Universal Robots PolyScope program: ability.urp

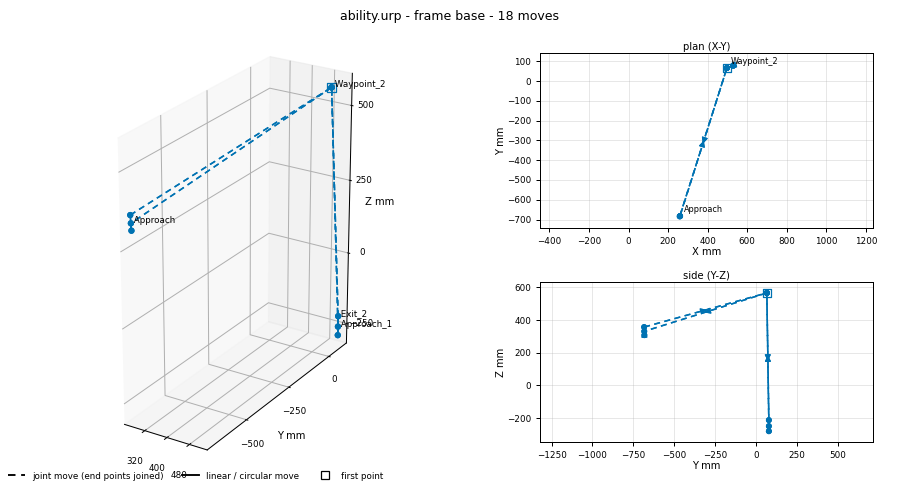
[picture p0: tool path of ability.urp in frame base, 18 of 18 moves have a stored position in this frame; points joined in program order, loops and branches not executed]
Program ability (installation=default directory=/programs createdIn=5.16.0 lastSavedIn=5.21.3 robotSerialNumber=20245590091)
Calibrated DH parameters: a=[0.000082, -0.206079, -0.372164, 0.000031, 0.000055, 0]; d=[0.162506, 220.320261, -282.089171, 61.902297, 0.099578, 0.098999]; alpha=[1.569879, -0.001688, 0.002003, 1.569052, -1.569943, 0]; deltaTheta=[0, -1.064762, 0.743886, 0.320883, 0.000002, 0]
InitVariablesNode variables(variable(name=Pallet_2_cnt_3, expression=1), variable(name=Pallet_2_cnt_4, expression=1), variable(name=Pallet_2_cnt_5, expression=1), variable(name=Pallet_2_cnt_6, expression=1), variable(name=Pallet_2_lct_3, expression=1), variable(name=Pallet_2_lct_4, expression=1), variable(name=Pallet_2_lct_5, expression=1), variable(name=Pallet_2_lct_6, expression=1), variable(name=Pallet_2_lno_3, expression=1), variable(name=Pallet_2_lno_4, expression=1), variable(name=Pallet_2_lno_5, expression=1), variable(name=Pallet_2_lno_6, expression=1), variable(name=Pallet_2_sep_3, expression=False), variable(name=Pallet_2_sep_4, expression=False), variable(name=Pallet_2_sep_5, expression=False), variable(name=Pallet_2_sep_6, expression=False), variable(name=Pallet_2_tct_3, expression=1), variable(name=Pallet_2_tct_4, expression=1), variable(name=Pallet_2_tct_5, expression=1), variable(name=Pallet_2_tct_6, expression=1), variable(name=qNearApproach, expression=[0,0,0,0,0,0]), variable(name=qNearApproach_1, expression=[0,0,0,0,0,0]), variable(name=qNearApproach_2, expression=[0,0,0,0,0,0]), variable(name=qNearApproach_3, expression=[0,0,0,0,0,0]))
Robot Program (runOnlyOnce=false)
  SafeHome (positionOptionType=SPEED_AND_ACCELERATION speed=1.047198 acceleration=1.396263 nextMotionTime=2)
  URCap ER-Ability (EnabledRobotics - ER-ABILITY, Enabled Robotics ApS)
    URCap EventNode (EnabledRobotics - ER-ABILITY, Enabled Robotics ApS) dataModel(er_eventnode_inpname=GripOpen, er_eventnode_retvalname=none)
      URCap Gripper (Robotiq_Grippers, Robotiq Inc.) dataModel(position=0.0, force=100.0, speed=100.0, positionInDouble=0.0, forceInDouble=100.0, speedInDouble=100.0, slaveIds=[9], blocking=true)
    URCap EventNode (EnabledRobotics - ER-ABILITY, Enabled Robotics ApS) dataModel(er_eventnode_inpname=GripClosed, er_eventnode_retvalname=none)
      URCap Gripper (Robotiq_Grippers, Robotiq Inc.) dataModel(position=100.0, force=70.0, speed=100.0, positionInDouble=100.0, forceInDouble=70.0, speedInDouble=100.0, slaveIds=[9], blocking=true)
    URCap EventNode (EnabledRobotics - ER-ABILITY, Enabled Robotics ApS) dataModel(er_eventnode_inpname=Unload, er_eventnode_retvalname=none, er_eventnode_input_arg_names=[arg_pose], er_eventnode_input_arg_types=[pose])
      Unload_ref := __er_Unload_arg_pose
      MoveJ speed 60 deg/s, acceleration 80 deg/s^2 (useActiveTCP=true optimoveEnabled=false optiMoveSpeed=0.3 optiMoveAcceleration=0.09) feature=Base
        Waypoint Waypoint_2: TCP in base x=497.545 y=66.443 z=565.568 mm, rx=2.1662 ry=-2.097 rz=-0.0588 rad; joints [173.064, -87.949, 75.071, -70.913, -94.278, -8.478] deg
      URCap Palletizing (polyscope-pallet-impl, Universal Robots) dataModel(palletFeature=Base, isPalletizing=true, Length(key=objectHeight value=0.02 unit=M), Variable(key=qNearApproach, variable(name=qNearApproach_1, initializeExpression=[0,0,0,0,0,0])), Variable(key=name, variable(name=Pallet_5)), Variable(key=globalCountingVariable, variable(name=Pallet_2_cnt_6, initializeExpression=1)), Variable(key=layerCountingVariable, variable(name=Pallet_2_lct_6, initializeExpression=1)), Variable(key=layerNumberVariable, variable(name=Pallet_2_lno_6, initializeExpression=1)), Variable(key=handleSeparatorVariable, variable(name=Pallet_2_sep_6, initializeExpression=False)), Variable(key=totalCountVariable, variable(name=Pallet_2_tct_6, initializeExpression=1)), Variable(key=referencePoint, variable(featureName=referencePoin_1)), Variable(key=separatorPoint, variable(featureName=separatorPoin_1))); state(isChildrenLocked=true)
        URCap Patterns (polyscope-pallet-impl, Universal Robots) state(isChildrenLocked=true)
          URCap Pattern (polyscope-pallet-impl, Universal Robots) dataModel(UUID=a5dc391e-8dfa-4d41-8d42-d1a3ee492412, patternType=LINE, objects=3, Variable(key=nameVariable, variable(name=Line_Pattern_7))); state(isChildrenLocked=true)
            URCap Item (polyscope-pallet-impl, Universal Robots) dataModel(UUID=72ff3311-31d3-41c2-b996-3017bdb4fd84, patternType=LINE, index=0, calibrationDeltaTheta=[-1.5094818129821053E-8, -1.0647624878232371, 0.7438857393498214, 0.32088328103969005, 1.7447632748163189E-6, 3.439939232040279E-7], calibrationA=[8.193426020278456E-5, -0.2060785642550941, -0.3721635571632287, 3.0822330236917175E-5, 5.5236874526065846E-5, 0.0], calibrationD=[0.1625058419451979, 220.32026122990015, -282.0891711692004, 61.90229668578863, 0.09957797525715827, 0.09899883734970352], calibrationAlpha=[1.569878535244303, -0.0016878983510277897, 0.002002552910479703, 1.5690521837938194, -1.5699432474464643, 0.0], calibrationJointChecksum=[-1471040491, -1470094786, -1472279970, -1460232730, -1457493897, -1460320911], calibrationStatus=2, calibrationValidChecksum=true, baseToFeature=[0.0, 0.0, 0.0, 0.0, 0.0, 0.0], TCPOffset=[-1.9242631868060522E-6, -1.9505851089895998E-7, -4.2845847764150236E-6, -5.771534998269337E-6, -3.203463145879142E-5, 1.411217115060646E-5], JointPositions(key=jointpositions, JointPosition(key=[1], Angle(key=pos value=3.039745 unit=RAD)), JointPosition(key=[2], Angle(key=pos value=-0.112207 unit=RAD)), JointPosition(key=[3], Angle(key=pos value=1.692084 unit=RAD)), JointPosition(key=[4], Angle(key=pos value=-3.160784 unit=RAD)), JointPosition(key=[5], Angle(key=pos value=-1.59557 unit=RAD)), JointPosition(key=[6], Angle(key=pos value=-0.133127 unit=RAD))), Variable(key=variable, variable(name=StartItem_7)))
            URCap Item (polyscope-pallet-impl, Universal Robots) dataModel(UUID=58fef9f4-1789-42d8-bc72-cd3fccb1f7d0, patternType=LINE, index=1, calibrationDeltaTheta=[-1.5094818129821053E-8, -1.0647624878232371, 0.7438857393498214, 0.32088328103969005, 1.7447632748163189E-6, 3.439939232040279E-7], calibrationA=[8.193426020278456E-5, -0.2060785642550941, -0.3721635571632287, 3.0822330236917175E-5, 5.5236874526065846E-5, 0.0], calibrationD=[0.1625058419451979, 220.32026122990015, -282.0891711692004, 61.90229668578863, 0.09957797525715827, 0.09899883734970352], calibrationAlpha=[1.569878535244303, -0.0016878983510277897, 0.002002552910479703, 1.5690521837938194, -1.5699432474464643, 0.0], calibrationJointChecksum=[-1471040491, -1470094786, -1472279970, -1460232730, -1457493897, -1460320911], calibrationStatus=2, calibrationValidChecksum=true, baseToFeature=[0.0, 0.0, 0.0, 0.0, 0.0, 0.0], TCPOffset=[6.884421240790917E-6, -1.3788864439701065E-5, -2.2303486297114983E-5, 3.976905791947326E-5, -9.131492742263298E-6, 1.144757581185306E-5], JointPositions(key=jointpositions, JointPosition(key=[1], Angle(key=pos value=2.706754 unit=RAD)), JointPosition(key=[2], Angle(key=pos value=-0.110768 unit=RAD)), JointPosition(key=[3], Angle(key=pos value=1.673712 unit=RAD)), JointPosition(key=[4], Angle(key=pos value=-3.151042 unit=RAD)), JointPosition(key=[5], Angle(key=pos value=-1.590635 unit=RAD)), JointPosition(key=[6], Angle(key=pos value=-0.466181 unit=RAD))), Variable(key=variable, variable(name=EndItem_7)))
        URCap Layers (polyscope-pallet-impl, Universal Robots) dataModel(separators=[false], selectedPatterns=[a5dc391e-8dfa-4d41-8d42-d1a3ee492412])
        URCap At Each Item (polyscope-pallet-impl, Universal Robots) dataModel(selectedPattern=a5dc391e-8dfa-4d41-8d42-d1a3ee492412, selectedPosition=72ff3311-31d3-41c2-b996-3017bdb4fd84, Approach_calibrationDeltaTheta=[-1.5094818129821053E-8, -1.0647624878232371, 0.7438857393498214, 0.32088328103969005, 1.7447632748163189E-6, 3.439939232040279E-7], Approach_calibrationA=[8.193426020278456E-5, -0.2060785642550941, -0.3721635571632287, 3.0822330236917175E-5, 5.5236874526065846E-5, 0.0], Approach_calibrationD=[0.1625058419451979, 220.32026122990015, -282.0891711692004, 61.90229668578863, 0.09957797525715827, 0.09899883734970352], Approach_calibrationAlpha=[1.569878535244303, -0.0016878983510277897, 0.002002552910479703, 1.5690521837938194, -1.5699432474464643, 0.0], Approach_calibrationJointChecksum=[-1471040491, -1470094786, -1472279970, -1460232730, -1457493897, -1460320911], Approach_calibrationStatus=2, Approach_calibrationValidChecksum=true, Approach_baseToFeature=[0.0, 0.0, 0.0, 0.0, 0.0, 0.0], Approach_TCPOffset=[-1.1739771630381313E-6, -5.9013202938773546E-6, 4.731632657406504E-6, 9.46543669298376E-6, -7.291023009343288E-6, -4.926571632538777E-6], Exit_calibrationDeltaTheta=[-1.5094818129821053E-8, -1.0647624878232371, 0.7438857393498214, 0.32088328103969005, 1.7447632748163189E-6, 3.439939232040279E-7], Exit_calibrationA=[8.193426020278456E-5, -0.2060785642550941, -0.3721635571632287, 3.0822330236917175E-5, 5.5236874526065846E-5, 0.0], Exit_calibrationD=[0.1625058419451979, 220.32026122990015, -282.0891711692004, 61.90229668578863, 0.09957797525715827, 0.09899883734970352], Exit_calibrationAlpha=[1.569878535244303, -0.0016878983510277897, 0.002002552910479703, 1.5690521837938194, -1.5699432474464643, 0.0], Exit_calibrationJointChecksum=[-1471040491, -1470094786, -1472279970, -1460232730, -1457493897, -1460320911], Exit_calibrationStatus=2, Exit_calibrationValidChecksum=true, Exit_baseToFeature=[0.0, 0.0, 0.0, 0.0, 0.0, 0.0], Exit_TCPOffset=[-1.296947476206456E-6, -4.670706427511995E-6, -4.147832971562737E-6, 1.5766715229967917E-6, -2.8354561647716597E-6, 2.251626105232425E-6], currentWizardState=LANDING, Pose(key=refBaseToFeature, Position(key=posePosition, Length(key=X value=0 unit=M), Length(key=Y value=0 unit=M), Length(key=Z value=0 unit=M)), Rotation(key=poseRotation, Angle(key=RX value=0 unit=RAD), Angle(key=RY value=0 unit=RAD), Angle(key=RZ value=0 unit=RAD))), Pose(key=refPose, Position(key=posePosition, Length(key=X value=0.529806 unit=M), Length(key=Y value=0.078793 unit=M), Length(key=Z value=-0.279912 unit=M)), Rotation(key=poseRotation, Angle(key=RX value=2.252769 unit=RAD), Angle(key=RY value=-2.172326 unit=RAD), Angle(key=RZ value=0.036579 unit=RAD))), JointPositions(key=Approach_jointpositions, JointPosition(key=[1], Angle(key=pos value=3.039864 unit=RAD)), JointPosition(key=[2], Angle(key=pos value=-0.185667 unit=RAD)), JointPosition(key=[3], Angle(key=pos value=1.753674 unit=RAD)), JointPosition(key=[4], Angle(key=pos value=-3.148901 unit=RAD)), JointPosition(key=[5], Angle(key=pos value=-1.595402 unit=RAD)), JointPosition(key=[6], Angle(key=pos value=-0.132955 unit=RAD))), JointPositions(key=Exit_jointpositions, JointPosition(key=[1], Angle(key=pos value=3.040007 unit=RAD)), JointPosition(key=[2], Angle(key=pos value=-0.275055 unit=RAD)), JointPosition(key=[3], Angle(key=pos value=1.820884 unit=RAD)), JointPosition(key=[4], Angle(key=pos value=-3.126719 unit=RAD)), JointPosition(key=[5], Angle(key=pos value=-1.595217 unit=RAD)), JointPosition(key=[6], Angle(key=pos value=-0.132784 unit=RAD))))
          URCap Generated Movements (polyscope-pallet-impl, Universal Robots) state(isChildrenLocked=true)
            MoveJ speed 60 deg/s, acceleration 80 deg/s^2 (useActiveTCP=true optimoveEnabled=false optiMoveSpeed=0.3 optiMoveAcceleration=0.09) feature=referencePoin_1
              Waypoint Approach_1: TCP in base x=529.812 y=78.794 z=-249.076 mm, rx=2.2528 ry=-2.1723 rz=0.0366 rad; joints [174.171, -10.638, 100.478, -180.419, -91.41, -7.618] deg; TCP offset x=-0.001 y=-0.006 z=0.005 mm, rx=0 ry=0 rz=0 rad; feature pose in base x=529.806 y=78.793 z=-279.912 mm, rx=2.2528 ry=-2.1723 rz=0.0366 rad
            MoveL speed 250 mm/s, acceleration 1200 mm/s^2 (useActiveTCP=true optimoveEnabled=false optiMoveSpeed=0.3 optiMoveAcceleration=0.09) feature(featureName=referencePoin_1)
              Waypoint ToolActionPoi_1: TCP in base x=529.806 y=78.793 z=-279.912 mm, rx=2.2528 ry=-2.1723 rz=0.0366 rad; joints [174.165, -6.429, 96.949, -181.1, -91.419, -7.628] deg; TCP offset x=-0.002 y=0 z=-0.004 mm, rx=0 ry=0 rz=0 rad
            Folder Tool action
              URCap Gripper (Robotiq_Grippers, Robotiq Inc.) dataModel(position=100.0, force=100.0, speed=100.0, positionInDouble=100.0, forceInDouble=100.0, speedInDouble=100.0, slaveIds=[9], blocking=true)
            MoveL speed 250 mm/s, acceleration 1200 mm/s^2 (useActiveTCP=true optimoveEnabled=false optiMoveSpeed=0.3 optiMoveAcceleration=0.09) feature(featureName=referencePoin_1)
              Waypoint Exit_2: TCP in base x=529.81 y=78.795 z=-211.983 mm, rx=2.2528 ry=-2.1723 rz=0.0366 rad; joints [174.18, -15.76, 104.329, -179.148, -91.399, -7.608] deg; TCP offset x=-0.001 y=-0.005 z=-0.004 mm, rx=0 ry=0 rz=0 rad
      MoveJ speed 60 deg/s, acceleration 80 deg/s^2 (useActiveTCP=true optimoveEnabled=false optiMoveSpeed=0.3 optiMoveAcceleration=0.09) feature=Base
        Waypoint Waypoint_2: TCP in base x=497.545 y=66.443 z=565.568 mm, rx=2.1662 ry=-2.097 rz=-0.0588 rad; joints [173.064, -87.949, 75.071, -70.913, -94.278, -8.478] deg
      URCap Palletizing (polyscope-pallet-impl, Universal Robots) dataModel(isPalletizing=true, palletFeature=Unload_ref, Length(key=objectHeight value=0.02 unit=M), Variable(key=qNearApproach, variable(name=qNearApproach_2, initializeExpression=[0,0,0,0,0,0])), Variable(key=name, variable(name=Pallet_1)), Variable(key=globalCountingVariable, variable(name=Pallet_2_cnt_5, initializeExpression=1)), Variable(key=layerCountingVariable, variable(name=Pallet_2_lct_5, initializeExpression=1)), Variable(key=layerNumberVariable, variable(name=Pallet_2_lno_5, initializeExpression=1)), Variable(key=handleSeparatorVariable, variable(name=Pallet_2_sep_5, initializeExpression=False)), Variable(key=totalCountVariable, variable(name=Pallet_2_tct_5, initializeExpression=1)), Variable(key=referencePoint, variable(featureName=referencePoin_2)), Variable(key=separatorPoint, variable(featureName=separatorPoin_2))); state(isChildrenLocked=true)
        URCap Patterns (polyscope-pallet-impl, Universal Robots) state(isChildrenLocked=true)
          URCap Pattern (polyscope-pallet-impl, Universal Robots) dataModel(UUID=07243d7f-bf8f-4104-9bd3-73f99270b9f6, patternType=LINE, objects=3, Variable(key=nameVariable, variable(name=Line_Pattern_1))); state(isChildrenLocked=true)
            URCap Item (polyscope-pallet-impl, Universal Robots) dataModel(UUID=e6243a9f-c885-4ed6-8873-203569e74fdc, patternType=LINE, index=0, calibrationDeltaTheta=[-1.5094818129821053E-8, -1.0647624878232371, 0.7438857393498214, 0.32088328103969005, 1.7447632748163189E-6, 3.439939232040279E-7], calibrationA=[8.193426020278456E-5, -0.2060785642550941, -0.3721635571632287, 3.0822330236917175E-5, 5.5236874526065846E-5, 0.0], calibrationD=[0.1625058419451979, 220.32026122990015, -282.0891711692004, 61.90229668578863, 0.09957797525715827, 0.09899883734970352], calibrationAlpha=[1.569878535244303, -0.0016878983510277897, 0.002002552910479703, 1.5690521837938194, -1.5699432474464643, 0.0], calibrationJointChecksum=[-1471040491, -1470094786, -1472279970, -1460232730, -1457493897, -1460320911], calibrationStatus=2, calibrationValidChecksum=true, baseToFeature=[0.3642472151847146, -0.6539896130686794, 0.3378929456834839, 0.09668575265698816, 3.0976550128318143, 0.04574427409651193], TCPOffset=[1.0537130964438646E-6, 3.1583842665661166E-6, -9.165165983537893E-6, 1.9395843013701872E-5, -1.1001609909023522E-5, 1.3091248772568936E-5], JointPositions(key=jointpositions, JointPosition(key=[1], Angle(key=pos value=1.744897 unit=RAD)), JointPosition(key=[2], Angle(key=pos value=-0.965579 unit=RAD)), JointPosition(key=[3], Angle(key=pos value=1.232646 unit=RAD)), JointPosition(key=[4], Angle(key=pos value=-1.816819 unit=RAD)), JointPosition(key=[5], Angle(key=pos value=-1.521721 unit=RAD)), JointPosition(key=[6], Angle(key=pos value=0.239107 unit=RAD))), Variable(key=variable, variable(name=StartItem_1)))
            URCap Item (polyscope-pallet-impl, Universal Robots) dataModel(UUID=c4ba0ccc-1ea8-4b4a-a0e5-b351c685b141, patternType=LINE, index=1, calibrationDeltaTheta=[-1.5094818129821053E-8, -1.0647624878232371, 0.7438857393498214, 0.32088328103969005, 1.7447632748163189E-6, 3.439939232040279E-7], calibrationA=[8.193426020278456E-5, -0.2060785642550941, -0.3721635571632287, 3.0822330236917175E-5, 5.5236874526065846E-5, 0.0], calibrationD=[0.1625058419451979, 220.32026122990015, -282.0891711692004, 61.90229668578863, 0.09957797525715827, 0.09899883734970352], calibrationAlpha=[1.569878535244303, -0.0016878983510277897, 0.002002552910479703, 1.5690521837938194, -1.5699432474464643, 0.0], calibrationJointChecksum=[-1471040491, -1470094786, -1472279970, -1460232730, -1457493897, -1460320911], calibrationStatus=2, calibrationValidChecksum=true, baseToFeature=[0.3642472151847146, -0.6539896130686794, 0.3378929456834839, 0.09668575265698816, 3.0976550128318143, 0.04574427409651193], TCPOffset=[-1.9181956956160207E-6, 3.271949199357138E-6, -1.0075163425771194E-6, -8.461158062938895E-6, 4.5656538735669615E-6, 3.0657126138548753E-6], JointPositions(key=jointpositions, JointPosition(key=[1], Angle(key=pos value=1.487256 unit=RAD)), JointPosition(key=[2], Angle(key=pos value=-1.092876 unit=RAD)), JointPosition(key=[3], Angle(key=pos value=1.431178 unit=RAD)), JointPosition(key=[4], Angle(key=pos value=-1.87667 unit=RAD)), JointPosition(key=[5], Angle(key=pos value=-1.528259 unit=RAD)), JointPosition(key=[6], Angle(key=pos value=-0.018683 unit=RAD))), Variable(key=variable, variable(name=EndItem_1)))
        URCap Layers (polyscope-pallet-impl, Universal Robots) dataModel(separators=[false], selectedPatterns=[07243d7f-bf8f-4104-9bd3-73f99270b9f6])
        URCap At Each Item (polyscope-pallet-impl, Universal Robots) dataModel(selectedPattern=07243d7f-bf8f-4104-9bd3-73f99270b9f6, selectedPosition=e6243a9f-c885-4ed6-8873-203569e74fdc, Approach_calibrationDeltaTheta=[-1.5094818129821053E-8, -1.0647624878232371, 0.7438857393498214, 0.32088328103969005, 1.7447632748163189E-6, 3.439939232040279E-7], Approach_calibrationA=[8.193426020278456E-5, -0.2060785642550941, -0.3721635571632287, 3.0822330236917175E-5, 5.5236874526065846E-5, 0.0], Approach_calibrationD=[0.1625058419451979, 220.32026122990015, -282.0891711692004, 61.90229668578863, 0.09957797525715827, 0.09899883734970352], Approach_calibrationAlpha=[1.569878535244303, -0.0016878983510277897, 0.002002552910479703, 1.5690521837938194, -1.5699432474464643, 0.0], Approach_calibrationJointChecksum=[-1471040491, -1470094786, -1472279970, -1460232730, -1457493897, -1460320911], Approach_calibrationStatus=2, Approach_calibrationValidChecksum=true, Approach_baseToFeature=[0.3642472151847146, -0.6539896130686794, 0.3378929456834839, 0.09668575265698816, 3.0976550128318143, 0.04574427409651193], Approach_TCPOffset=[4.38855060347354E-6, -4.899361530807944E-6, 2.8712706818478928E-5, -3.3818317639434483E-5, -1.9006392708885734E-6, -4.541078720377721E-6], Exit_calibrationDeltaTheta=[-1.5094818129821053E-8, -1.0647624878232371, 0.7438857393498214, 0.32088328103969005, 1.7447632748163189E-6, 3.439939232040279E-7], Exit_calibrationA=[8.193426020278456E-5, -0.2060785642550941, -0.3721635571632287, 3.0822330236917175E-5, 5.5236874526065846E-5, 0.0], Exit_calibrationD=[0.1625058419451979, 220.32026122990015, -282.0891711692004, 61.90229668578863, 0.09957797525715827, 0.09899883734970352], Exit_calibrationAlpha=[1.569878535244303, -0.0016878983510277897, 0.002002552910479703, 1.5690521837938194, -1.5699432474464643, 0.0], Exit_calibrationJointChecksum=[-1471040491, -1470094786, -1472279970, -1460232730, -1457493897, -1460320911], Exit_calibrationStatus=2, Exit_calibrationValidChecksum=true, Exit_baseToFeature=[0.3642472151847146, -0.6539896130686794, 0.3378929456834839, 0.09668575265698816, 3.0976550128318143, 0.04574427409651193], Exit_TCPOffset=[-2.261881683229827E-6, -6.1489387452873245E-6, 3.387991530712231E-6, 6.960322118020412E-6, -3.138926643113733E-5, 1.113853935195239E-5], currentWizardState=LANDING, Pose(key=refBaseToFeature, Position(key=posePosition, Length(key=X value=0.364247 unit=M), Length(key=Y value=-0.65399 unit=M), Length(key=Z value=0.337893 unit=M)), Rotation(key=poseRotation, Angle(key=RX value=0.096686 unit=RAD), Angle(key=RY value=3.097655 unit=RAD), Angle(key=RZ value=0.045744 unit=RAD))), Pose(key=refPose, Position(key=posePosition, Length(key=X value=0.260951 unit=M), Length(key=Y value=-0.682557 unit=M), Length(key=Z value=0.307415 unit=M)), Rotation(key=poseRotation, Angle(key=RX value=0.09672 unit=RAD), Angle(key=RY value=3.097651 unit=RAD), Angle(key=RZ value=0.045742 unit=RAD))), JointPositions(key=Approach_jointpositions, JointPosition(key=[1], Angle(key=pos value=1.743379 unit=RAD)), JointPosition(key=[2], Angle(key=pos value=-0.978991 unit=RAD)), JointPosition(key=[3], Angle(key=pos value=1.192911 unit=RAD)), JointPosition(key=[4], Angle(key=pos value=-1.763616 unit=RAD)), JointPosition(key=[5], Angle(key=pos value=-1.521736 unit=RAD)), JointPosition(key=[6], Angle(key=pos value=0.237484 unit=RAD))), JointPositions(key=Exit_jointpositions, JointPosition(key=[1], Angle(key=pos value=1.741694 unit=RAD)), JointPosition(key=[2], Angle(key=pos value=-0.990422 unit=RAD)), JointPosition(key=[3], Angle(key=pos value=1.143754 unit=RAD)), JointPosition(key=[4], Angle(key=pos value=-1.702942 unit=RAD)), JointPosition(key=[5], Angle(key=pos value=-1.521773 unit=RAD)), JointPosition(key=[6], Angle(key=pos value=0.235669 unit=RAD))))
          URCap Generated Movements (polyscope-pallet-impl, Universal Robots) state(isChildrenLocked=true)
            MoveJ speed 60 deg/s, acceleration 80 deg/s^2 (useActiveTCP=true optimoveEnabled=false optiMoveSpeed=0.3 optiMoveAcceleration=0.09) feature=referencePoin_2
              Waypoint Approach: TCP in base x=259.939 y=-683.222 z=330.824 mm, rx=0.0967 ry=3.0976 rz=0.0458 rad; joints [99.888, -56.092, 68.349, -101.048, -87.189, 13.607] deg; TCP offset x=0.004 y=-0.005 z=0.029 mm, rx=0 ry=0 rz=0 rad; feature pose in base x=260.951 y=-682.557 z=307.415 mm, rx=0.0967 ry=3.0977 rz=0.0457 rad
            MoveL speed 250 mm/s, acceleration 1200 mm/s^2 (useActiveTCP=true optimoveEnabled=false optiMoveSpeed=0.3 optiMoveAcceleration=0.09) feature(featureName=referencePoin_2)
              Waypoint ToolActionPoint: TCP in base x=260.951 y=-682.557 z=307.415 mm, rx=0.0967 ry=3.0977 rz=0.0457 rad; joints [99.975, -55.324, 70.625, -104.096, -87.188, 13.7] deg; TCP offset x=0.001 y=0.003 z=-0.009 mm, rx=0 ry=0 rz=0 rad
            Folder Tool action
              URCap Gripper (Robotiq_Grippers, Robotiq Inc.) dataModel(position=0.0, force=100.0, speed=100.0, positionInDouble=0.0, forceInDouble=100.0, speedInDouble=100.0, slaveIds=[9], blocking=true)
            MoveL speed 250 mm/s, acceleration 1200 mm/s^2 (useActiveTCP=true optimoveEnabled=false optiMoveSpeed=0.3 optiMoveAcceleration=0.09) feature(featureName=referencePoin_2)
              Waypoint Exit_1: TCP in base x=258.824 y=-683.959 z=356.887 mm, rx=0.0967 ry=3.0976 rz=0.0457 rad; joints [99.792, -56.747, 65.532, -97.571, -87.191, 13.503] deg; TCP offset x=-0.002 y=-0.006 z=0.003 mm, rx=0 ry=0 rz=0 rad
      MoveJ speed 60 deg/s, acceleration 80 deg/s^2 (useActiveTCP=true optimoveEnabled=false optiMoveSpeed=0.3 optiMoveAcceleration=0.09) feature=Base
        Waypoint Waypoint_2: TCP in base x=497.545 y=66.443 z=565.568 mm, rx=2.1662 ry=-2.097 rz=-0.0588 rad; joints [173.064, -87.949, 75.071, -70.913, -94.278, -8.478] deg
    URCap EventNode (EnabledRobotics - ER-ABILITY, Enabled Robotics ApS) dataModel(er_eventnode_inpname=Palletize, er_eventnode_retvalname=none, er_eventnode_input_arg_names=[arg_pose], er_eventnode_input_arg_types=[pose])
      Pallet_ref := __er_Palletize_arg_pose
      MoveJ speed 60 deg/s, acceleration 80 deg/s^2 (useActiveTCP=true optimoveEnabled=false optiMoveSpeed=0.3 optiMoveAcceleration=0.09) feature=Base
        Waypoint Waypoint_2: TCP in base x=497.545 y=66.443 z=565.568 mm, rx=2.1662 ry=-2.097 rz=-0.0588 rad; joints [173.064, -87.949, 75.071, -70.913, -94.278, -8.478] deg
      URCap Palletizing (polyscope-pallet-impl, Universal Robots) dataModel(isPalletizing=true, palletFeature=Pallet_ref, Length(key=objectHeight value=0.02 unit=M), Variable(key=qNearApproach, variable(name=qNearApproach, initializeExpression=[0,0,0,0,0,0])), Variable(key=name, variable(name=Pallet_3)), Variable(key=globalCountingVariable, variable(name=Pallet_2_cnt_3, initializeExpression=1)), Variable(key=layerCountingVariable, variable(name=Pallet_2_lct_3, initializeExpression=1)), Variable(key=layerNumberVariable, variable(name=Pallet_2_lno_3, initializeExpression=1)), Variable(key=handleSeparatorVariable, variable(name=Pallet_2_sep_3, initializeExpression=False)), Variable(key=totalCountVariable, variable(name=Pallet_2_tct_3, initializeExpression=1)), Variable(key=referencePoint, variable(featureName=referencePoin_3)), Variable(key=separatorPoint, variable(featureName=separatorPoin_3))); state(isChildrenLocked=true)
        URCap Patterns (polyscope-pallet-impl, Universal Robots) state(isChildrenLocked=true)
          URCap Pattern (polyscope-pallet-impl, Universal Robots) dataModel(UUID=07243d7f-bf8f-4104-9bd3-73f99270b9f6, patternType=LINE, objects=3, Variable(key=nameVariable, variable(name=Line_Pattern_5))); state(isChildrenLocked=true)
            URCap Item (polyscope-pallet-impl, Universal Robots) dataModel(UUID=e6243a9f-c885-4ed6-8873-203569e74fdc, patternType=LINE, index=0, calibrationDeltaTheta=[-1.5094818129821053E-8, -1.0647624878232371, 0.7438857393498214, 0.32088328103969005, 1.7447632748163189E-6, 3.439939232040279E-7], calibrationA=[8.193426020278456E-5, -0.2060785642550941, -0.3721635571632287, 3.0822330236917175E-5, 5.5236874526065846E-5, 0.0], calibrationD=[0.1625058419451979, 220.32026122990015, -282.0891711692004, 61.90229668578863, 0.09957797525715827, 0.09899883734970352], calibrationAlpha=[1.569878535244303, -0.0016878983510277897, 0.002002552910479703, 1.5690521837938194, -1.5699432474464643, 0.0], calibrationJointChecksum=[-1471040491, -1470094786, -1472279970, -1460232730, -1457493897, -1460320911], calibrationStatus=2, calibrationValidChecksum=true, baseToFeature=[0.3642472151847146, -0.6539896130686794, 0.3378929456834839, 0.09668575265698816, 3.0976550128318143, 0.04574427409651193], TCPOffset=[1.0537130964438646E-6, 3.1583842665661166E-6, -9.165165983537893E-6, 1.9395843013701872E-5, -1.1001609909023522E-5, 1.3091248772568936E-5], JointPositions(key=jointpositions, JointPosition(key=[1], Angle(key=pos value=1.744897 unit=RAD)), JointPosition(key=[2], Angle(key=pos value=-0.965579 unit=RAD)), JointPosition(key=[3], Angle(key=pos value=1.232646 unit=RAD)), JointPosition(key=[4], Angle(key=pos value=-1.816819 unit=RAD)), JointPosition(key=[5], Angle(key=pos value=-1.521721 unit=RAD)), JointPosition(key=[6], Angle(key=pos value=0.239107 unit=RAD))), Variable(key=variable, variable(name=StartItem_5)))
            URCap Item (polyscope-pallet-impl, Universal Robots) dataModel(UUID=c4ba0ccc-1ea8-4b4a-a0e5-b351c685b141, patternType=LINE, index=1, calibrationDeltaTheta=[-1.5094818129821053E-8, -1.0647624878232371, 0.7438857393498214, 0.32088328103969005, 1.7447632748163189E-6, 3.439939232040279E-7], calibrationA=[8.193426020278456E-5, -0.2060785642550941, -0.3721635571632287, 3.0822330236917175E-5, 5.5236874526065846E-5, 0.0], calibrationD=[0.1625058419451979, 220.32026122990015, -282.0891711692004, 61.90229668578863, 0.09957797525715827, 0.09899883734970352], calibrationAlpha=[1.569878535244303, -0.0016878983510277897, 0.002002552910479703, 1.5690521837938194, -1.5699432474464643, 0.0], calibrationJointChecksum=[-1471040491, -1470094786, -1472279970, -1460232730, -1457493897, -1460320911], calibrationStatus=2, calibrationValidChecksum=true, baseToFeature=[0.3642472151847146, -0.6539896130686794, 0.3378929456834839, 0.09668575265698816, 3.0976550128318143, 0.04574427409651193], TCPOffset=[-1.9181956956160207E-6, 3.271949199357138E-6, -1.0075163425771194E-6, -8.461158062938895E-6, 4.5656538735669615E-6, 3.0657126138548753E-6], JointPositions(key=jointpositions, JointPosition(key=[1], Angle(key=pos value=1.487256 unit=RAD)), JointPosition(key=[2], Angle(key=pos value=-1.092876 unit=RAD)), JointPosition(key=[3], Angle(key=pos value=1.431178 unit=RAD)), JointPosition(key=[4], Angle(key=pos value=-1.87667 unit=RAD)), JointPosition(key=[5], Angle(key=pos value=-1.528259 unit=RAD)), JointPosition(key=[6], Angle(key=pos value=-0.018683 unit=RAD))), Variable(key=variable, variable(name=EndItem_5)))
        URCap Layers (polyscope-pallet-impl, Universal Robots) dataModel(separators=[false], selectedPatterns=[07243d7f-bf8f-4104-9bd3-73f99270b9f6])
        URCap At Each Item (polyscope-pallet-impl, Universal Robots) dataModel(selectedPattern=07243d7f-bf8f-4104-9bd3-73f99270b9f6, selectedPosition=e6243a9f-c885-4ed6-8873-203569e74fdc, Approach_calibrationDeltaTheta=[-1.5094818129821053E-8, -1.0647624878232371, 0.7438857393498214, 0.32088328103969005, 1.7447632748163189E-6, 3.439939232040279E-7], Approach_calibrationA=[8.193426020278456E-5, -0.2060785642550941, -0.3721635571632287, 3.0822330236917175E-5, 5.5236874526065846E-5, 0.0], Approach_calibrationD=[0.1625058419451979, 220.32026122990015, -282.0891711692004, 61.90229668578863, 0.09957797525715827, 0.09899883734970352], Approach_calibrationAlpha=[1.569878535244303, -0.0016878983510277897, 0.002002552910479703, 1.5690521837938194, -1.5699432474464643, 0.0], Approach_calibrationJointChecksum=[-1471040491, -1470094786, -1472279970, -1460232730, -1457493897, -1460320911], Approach_calibrationStatus=2, Approach_calibrationValidChecksum=true, Approach_baseToFeature=[0.3642472151847146, -0.6539896130686794, 0.3378929456834839, 0.09668575265698816, 3.0976550128318143, 0.04574427409651193], Approach_TCPOffset=[4.38855060347354E-6, -4.899361530807944E-6, 2.8712706818478928E-5, -3.3818317639434483E-5, -1.9006392708885734E-6, -4.541078720377721E-6], Exit_calibrationDeltaTheta=[-1.5094818129821053E-8, -1.0647624878232371, 0.7438857393498214, 0.32088328103969005, 1.7447632748163189E-6, 3.439939232040279E-7], Exit_calibrationA=[8.193426020278456E-5, -0.2060785642550941, -0.3721635571632287, 3.0822330236917175E-5, 5.5236874526065846E-5, 0.0], Exit_calibrationD=[0.1625058419451979, 220.32026122990015, -282.0891711692004, 61.90229668578863, 0.09957797525715827, 0.09899883734970352], Exit_calibrationAlpha=[1.569878535244303, -0.0016878983510277897, 0.002002552910479703, 1.5690521837938194, -1.5699432474464643, 0.0], Exit_calibrationJointChecksum=[-1471040491, -1470094786, -1472279970, -1460232730, -1457493897, -1460320911], Exit_calibrationStatus=2, Exit_calibrationValidChecksum=true, Exit_baseToFeature=[0.3642472151847146, -0.6539896130686794, 0.3378929456834839, 0.09668575265698816, 3.0976550128318143, 0.04574427409651193], Exit_TCPOffset=[-2.261881683229827E-6, -6.1489387452873245E-6, 3.387991530712231E-6, 6.960322118020412E-6, -3.138926643113733E-5, 1.113853935195239E-5], currentWizardState=LANDING, Pose(key=refBaseToFeature, Position(key=posePosition, Length(key=X value=0.364247 unit=M), Length(key=Y value=-0.65399 unit=M), Length(key=Z value=0.337893 unit=M)), Rotation(key=poseRotation, Angle(key=RX value=0.096686 unit=RAD), Angle(key=RY value=3.097655 unit=RAD), Angle(key=RZ value=0.045744 unit=RAD))), Pose(key=refPose, Position(key=posePosition, Length(key=X value=0.260951 unit=M), Length(key=Y value=-0.682557 unit=M), Length(key=Z value=0.307415 unit=M)), Rotation(key=poseRotation, Angle(key=RX value=0.09672 unit=RAD), Angle(key=RY value=3.097651 unit=RAD), Angle(key=RZ value=0.045742 unit=RAD))), JointPositions(key=Approach_jointpositions, JointPosition(key=[1], Angle(key=pos value=1.743379 unit=RAD)), JointPosition(key=[2], Angle(key=pos value=-0.978991 unit=RAD)), JointPosition(key=[3], Angle(key=pos value=1.192911 unit=RAD)), JointPosition(key=[4], Angle(key=pos value=-1.763616 unit=RAD)), JointPosition(key=[5], Angle(key=pos value=-1.521736 unit=RAD)), JointPosition(key=[6], Angle(key=pos value=0.237484 unit=RAD))), JointPositions(key=Exit_jointpositions, JointPosition(key=[1], Angle(key=pos value=1.741694 unit=RAD)), JointPosition(key=[2], Angle(key=pos value=-0.990422 unit=RAD)), JointPosition(key=[3], Angle(key=pos value=1.143754 unit=RAD)), JointPosition(key=[4], Angle(key=pos value=-1.702942 unit=RAD)), JointPosition(key=[5], Angle(key=pos value=-1.521773 unit=RAD)), JointPosition(key=[6], Angle(key=pos value=0.235669 unit=RAD))))
          URCap Generated Movements (polyscope-pallet-impl, Universal Robots) state(isChildrenLocked=true)
            MoveJ speed 60 deg/s, acceleration 80 deg/s^2 (useActiveTCP=false optimoveEnabled=false optiMoveSpeed=0.3 optiMoveAcceleration=0.09) tcp=TCP; feature=referencePoin_3
              Waypoint Approach: TCP in base x=259.939 y=-683.222 z=330.824 mm, rx=0.0967 ry=3.0976 rz=0.0458 rad; joints [99.888, -56.092, 68.349, -101.048, -87.189, 13.607] deg; TCP offset x=0.004 y=-0.005 z=0.029 mm, rx=0 ry=0 rz=0 rad; feature pose in base x=260.951 y=-682.557 z=307.415 mm, rx=0.0967 ry=3.0977 rz=0.0457 rad
            MoveL speed 250 mm/s, acceleration 1200 mm/s^2 (useActiveTCP=true optimoveEnabled=false optiMoveSpeed=0.3 optiMoveAcceleration=0.09) feature=referencePoin_3
              Waypoint ToolActionPoint: TCP in base x=260.951 y=-682.557 z=307.415 mm, rx=0.0967 ry=3.0977 rz=0.0457 rad; joints [99.975, -55.324, 70.625, -104.096, -87.188, 13.7] deg; TCP offset x=0.001 y=0.003 z=-0.009 mm, rx=0 ry=0 rz=0 rad
            Folder Tool action
              URCap Gripper (Robotiq_Grippers, Robotiq Inc.) dataModel(position=100.0, force=0.0, speed=98.0, positionInDouble=100.0, forceInDouble=0.0, speedInDouble=98.0, slaveIds=[9], blocking=true)
            MoveL speed 250 mm/s, acceleration 1200 mm/s^2 (useActiveTCP=true optimoveEnabled=false optiMoveSpeed=0.3 optiMoveAcceleration=0.09) feature=referencePoin_3
              Waypoint Exit_1: TCP in base x=258.824 y=-683.959 z=356.887 mm, rx=0.0967 ry=3.0976 rz=0.0457 rad; joints [99.792, -56.747, 65.532, -97.571, -87.191, 13.503] deg; TCP offset x=-0.002 y=-0.006 z=0.003 mm, rx=0 ry=0 rz=0 rad
      MoveJ speed 60 deg/s, acceleration 80 deg/s^2 (useActiveTCP=true optimoveEnabled=false optiMoveSpeed=0.3 optiMoveAcceleration=0.09) feature=Base
        Waypoint Waypoint_2: TCP in base x=497.545 y=66.443 z=565.568 mm, rx=2.1662 ry=-2.097 rz=-0.0588 rad; joints [173.064, -87.949, 75.071, -70.913, -94.278, -8.478] deg
      URCap Palletizing (polyscope-pallet-impl, Universal Robots) dataModel(palletFeature=Base, isPalletizing=true, Length(key=objectHeight value=0.02 unit=M), Variable(key=qNearApproach, variable(name=qNearApproach_3, initializeExpression=[0,0,0,0,0,0])), Variable(key=name, variable(name=Pallet_4)), Variable(key=globalCountingVariable, variable(name=Pallet_2_cnt_4, initializeExpression=1)), Variable(key=layerCountingVariable, variable(name=Pallet_2_lct_4, initializeExpression=1)), Variable(key=layerNumberVariable, variable(name=Pallet_2_lno_4, initializeExpression=1)), Variable(key=handleSeparatorVariable, variable(name=Pallet_2_sep_4, initializeExpression=False)), Variable(key=totalCountVariable, variable(name=Pallet_2_tct_4, initializeExpression=1)), Variable(key=referencePoint, variable(featureName=referencePoin_4)), Variable(key=separatorPoint, variable(featureName=separatorPoin_4))); state(isChildrenLocked=true)
        URCap Patterns (polyscope-pallet-impl, Universal Robots) state(isChildrenLocked=true)
          URCap Pattern (polyscope-pallet-impl, Universal Robots) dataModel(UUID=a5dc391e-8dfa-4d41-8d42-d1a3ee492412, patternType=LINE, objects=3, Variable(key=nameVariable, variable(name=Line_Pattern_6))); state(isChildrenLocked=true)
            URCap Item (polyscope-pallet-impl, Universal Robots) dataModel(UUID=72ff3311-31d3-41c2-b996-3017bdb4fd84, patternType=LINE, index=0, calibrationDeltaTheta=[-1.5094818129821053E-8, -1.0647624878232371, 0.7438857393498214, 0.32088328103969005, 1.7447632748163189E-6, 3.439939232040279E-7], calibrationA=[8.193426020278456E-5, -0.2060785642550941, -0.3721635571632287, 3.0822330236917175E-5, 5.5236874526065846E-5, 0.0], calibrationD=[0.1625058419451979, 220.32026122990015, -282.0891711692004, 61.90229668578863, 0.09957797525715827, 0.09899883734970352], calibrationAlpha=[1.569878535244303, -0.0016878983510277897, 0.002002552910479703, 1.5690521837938194, -1.5699432474464643, 0.0], calibrationJointChecksum=[-1471040491, -1470094786, -1472279970, -1460232730, -1457493897, -1460320911], calibrationStatus=2, calibrationValidChecksum=true, baseToFeature=[0.0, 0.0, 0.0, 0.0, 0.0, 0.0], TCPOffset=[-1.9242631868060522E-6, -1.9505851089895998E-7, -4.2845847764150236E-6, -5.771534998269337E-6, -3.203463145879142E-5, 1.411217115060646E-5], JointPositions(key=jointpositions, JointPosition(key=[1], Angle(key=pos value=3.039745 unit=RAD)), JointPosition(key=[2], Angle(key=pos value=-0.112207 unit=RAD)), JointPosition(key=[3], Angle(key=pos value=1.692084 unit=RAD)), JointPosition(key=[4], Angle(key=pos value=-3.160784 unit=RAD)), JointPosition(key=[5], Angle(key=pos value=-1.59557 unit=RAD)), JointPosition(key=[6], Angle(key=pos value=-0.133127 unit=RAD))), Variable(key=variable, variable(name=StartItem_6)))
            URCap Item (polyscope-pallet-impl, Universal Robots) dataModel(UUID=58fef9f4-1789-42d8-bc72-cd3fccb1f7d0, patternType=LINE, index=1, calibrationDeltaTheta=[-1.5094818129821053E-8, -1.0647624878232371, 0.7438857393498214, 0.32088328103969005, 1.7447632748163189E-6, 3.439939232040279E-7], calibrationA=[8.193426020278456E-5, -0.2060785642550941, -0.3721635571632287, 3.0822330236917175E-5, 5.5236874526065846E-5, 0.0], calibrationD=[0.1625058419451979, 220.32026122990015, -282.0891711692004, 61.90229668578863, 0.09957797525715827, 0.09899883734970352], calibrationAlpha=[1.569878535244303, -0.0016878983510277897, 0.002002552910479703, 1.5690521837938194, -1.5699432474464643, 0.0], calibrationJointChecksum=[-1471040491, -1470094786, -1472279970, -1460232730, -1457493897, -1460320911], calibrationStatus=2, calibrationValidChecksum=true, baseToFeature=[0.0, 0.0, 0.0, 0.0, 0.0, 0.0], TCPOffset=[6.884421240790917E-6, -1.3788864439701065E-5, -2.2303486297114983E-5, 3.976905791947326E-5, -9.131492742263298E-6, 1.144757581185306E-5], JointPositions(key=jointpositions, JointPosition(key=[1], Angle(key=pos value=2.706754 unit=RAD)), JointPosition(key=[2], Angle(key=pos value=-0.110768 unit=RAD)), JointPosition(key=[3], Angle(key=pos value=1.673712 unit=RAD)), JointPosition(key=[4], Angle(key=pos value=-3.151042 unit=RAD)), JointPosition(key=[5], Angle(key=pos value=-1.590635 unit=RAD)), JointPosition(key=[6], Angle(key=pos value=-0.466181 unit=RAD))), Variable(key=variable, variable(name=EndItem_6)))
        URCap Layers (polyscope-pallet-impl, Universal Robots) dataModel(separators=[false], selectedPatterns=[a5dc391e-8dfa-4d41-8d42-d1a3ee492412])
        URCap At Each Item (polyscope-pallet-impl, Universal Robots) dataModel(selectedPattern=a5dc391e-8dfa-4d41-8d42-d1a3ee492412, selectedPosition=72ff3311-31d3-41c2-b996-3017bdb4fd84, Approach_calibrationDeltaTheta=[-1.5094818129821053E-8, -1.0647624878232371, 0.7438857393498214, 0.32088328103969005, 1.7447632748163189E-6, 3.439939232040279E-7], Approach_calibrationA=[8.193426020278456E-5, -0.2060785642550941, -0.3721635571632287, 3.0822330236917175E-5, 5.5236874526065846E-5, 0.0], Approach_calibrationD=[0.1625058419451979, 220.32026122990015, -282.0891711692004, 61.90229668578863, 0.09957797525715827, 0.09899883734970352], Approach_calibrationAlpha=[1.569878535244303, -0.0016878983510277897, 0.002002552910479703, 1.5690521837938194, -1.5699432474464643, 0.0], Approach_calibrationJointChecksum=[-1471040491, -1470094786, -1472279970, -1460232730, -1457493897, -1460320911], Approach_calibrationStatus=2, Approach_calibrationValidChecksum=true, Approach_baseToFeature=[0.0, 0.0, 0.0, 0.0, 0.0, 0.0], Approach_TCPOffset=[-1.1739771630381313E-6, -5.9013202938773546E-6, 4.731632657406504E-6, 9.46543669298376E-6, -7.291023009343288E-6, -4.926571632538777E-6], Exit_calibrationDeltaTheta=[-1.5094818129821053E-8, -1.0647624878232371, 0.7438857393498214, 0.32088328103969005, 1.7447632748163189E-6, 3.439939232040279E-7], Exit_calibrationA=[8.193426020278456E-5, -0.2060785642550941, -0.3721635571632287, 3.0822330236917175E-5, 5.5236874526065846E-5, 0.0], Exit_calibrationD=[0.1625058419451979, 220.32026122990015, -282.0891711692004, 61.90229668578863, 0.09957797525715827, 0.09899883734970352], Exit_calibrationAlpha=[1.569878535244303, -0.0016878983510277897, 0.002002552910479703, 1.5690521837938194, -1.5699432474464643, 0.0], Exit_calibrationJointChecksum=[-1471040491, -1470094786, -1472279970, -1460232730, -1457493897, -1460320911], Exit_calibrationStatus=2, Exit_calibrationValidChecksum=true, Exit_baseToFeature=[0.0, 0.0, 0.0, 0.0, 0.0, 0.0], Exit_TCPOffset=[-1.296947476206456E-6, -4.670706427511995E-6, -4.147832971562737E-6, 1.5766715229967917E-6, -2.8354561647716597E-6, 2.251626105232425E-6], currentWizardState=LANDING, Pose(key=refBaseToFeature, Position(key=posePosition, Length(key=X value=0 unit=M), Length(key=Y value=0 unit=M), Length(key=Z value=0 unit=M)), Rotation(key=poseRotation, Angle(key=RX value=0 unit=RAD), Angle(key=RY value=0 unit=RAD), Angle(key=RZ value=0 unit=RAD))), Pose(key=refPose, Position(key=posePosition, Length(key=X value=0.529806 unit=M), Length(key=Y value=0.078793 unit=M), Length(key=Z value=-0.279912 unit=M)), Rotation(key=poseRotation, Angle(key=RX value=2.252769 unit=RAD), Angle(key=RY value=-2.172326 unit=RAD), Angle(key=RZ value=0.036579 unit=RAD))), JointPositions(key=Approach_jointpositions, JointPosition(key=[1], Angle(key=pos value=3.039864 unit=RAD)), JointPosition(key=[2], Angle(key=pos value=-0.185667 unit=RAD)), JointPosition(key=[3], Angle(key=pos value=1.753674 unit=RAD)), JointPosition(key=[4], Angle(key=pos value=-3.148901 unit=RAD)), JointPosition(key=[5], Angle(key=pos value=-1.595402 unit=RAD)), JointPosition(key=[6], Angle(key=pos value=-0.132955 unit=RAD))), JointPositions(key=Exit_jointpositions, JointPosition(key=[1], Angle(key=pos value=3.040007 unit=RAD)), JointPosition(key=[2], Angle(key=pos value=-0.275055 unit=RAD)), JointPosition(key=[3], Angle(key=pos value=1.820884 unit=RAD)), JointPosition(key=[4], Angle(key=pos value=-3.126719 unit=RAD)), JointPosition(key=[5], Angle(key=pos value=-1.595217 unit=RAD)), JointPosition(key=[6], Angle(key=pos value=-0.132784 unit=RAD))))
          URCap Generated Movements (polyscope-pallet-impl, Universal Robots) state(isChildrenLocked=true)
            MoveJ speed 60 deg/s, acceleration 80 deg/s^2 (useActiveTCP=true optimoveEnabled=false optiMoveSpeed=0.3 optiMoveAcceleration=0.09) feature=referencePoin_4
              Waypoint Approach_1: TCP in base x=529.812 y=78.794 z=-249.076 mm, rx=2.2528 ry=-2.1723 rz=0.0366 rad; joints [174.171, -10.638, 100.478, -180.419, -91.41, -7.618] deg; TCP offset x=-0.001 y=-0.006 z=0.005 mm, rx=0 ry=0 rz=0 rad; feature pose in base x=529.806 y=78.793 z=-279.912 mm, rx=2.2528 ry=-2.1723 rz=0.0366 rad
            MoveL speed 250 mm/s, acceleration 1200 mm/s^2 (useActiveTCP=true optimoveEnabled=false optiMoveSpeed=0.3 optiMoveAcceleration=0.09) feature=referencePoin_4
              Waypoint ToolActionPoi_1: TCP in base x=529.806 y=78.793 z=-279.912 mm, rx=2.2528 ry=-2.1723 rz=0.0366 rad; joints [174.165, -6.429, 96.949, -181.1, -91.419, -7.628] deg; TCP offset x=-0.002 y=0 z=-0.004 mm, rx=0 ry=0 rz=0 rad
            Folder Tool action
              URCap Gripper (Robotiq_Grippers, Robotiq Inc.) dataModel(position=0.0, force=0.0, speed=98.0, positionInDouble=0.0, forceInDouble=0.0, speedInDouble=98.0, slaveIds=[9], blocking=true)
            MoveL speed 250 mm/s, acceleration 1200 mm/s^2 (useActiveTCP=true optimoveEnabled=false optiMoveSpeed=0.3 optiMoveAcceleration=0.09) feature=referencePoin_4
              Waypoint Exit_2: TCP in base x=529.81 y=78.795 z=-211.983 mm, rx=2.2528 ry=-2.1723 rz=0.0366 rad; joints [174.18, -15.76, 104.329, -179.148, -91.399, -7.608] deg; TCP offset x=-0.001 y=-0.005 z=-0.004 mm, rx=0 ry=0 rz=0 rad
      MoveJ speed 60 deg/s, acceleration 80 deg/s^2 (useActiveTCP=true optimoveEnabled=false optiMoveSpeed=0.3 optiMoveAcceleration=0.09) feature=Base
        Waypoint Waypoint_2: TCP in base x=497.545 y=66.443 z=565.568 mm, rx=2.1662 ry=-2.097 rz=-0.0588 rad; joints [173.064, -87.949, 75.071, -70.913, -94.278, -8.478] deg
